ABB RAPID module: RsTempModule.mod

MODULE RsTempModule
    LOCAL CONST robtarget Target_10:=[[1336,100,940],[0.180407894,-0.26458531,0.050458418,0.945992364],[0,0,0,0],[9E+09,9E+09,9E+09,9E+09,9E+09,9E+09]];
    LOCAL CONST robtarget Target_20:=[[1131.146597498,-0.535735061,989.137836506],[0.652828066,-0.271690111,-0.271690111,-0.652828066],[0,0,0,0],[9E+09,9E+09,9E+09,9E+09,9E+09,9E+09]];
    LOCAL CONST robtarget Target_30:=[[1336,-49,1090],[0.946229257,-0.045801741,0.154506016,0.280500063],[0,0,0,0],[9E+09,9E+09,9E+09,9E+09,9E+09,9E+09]];
PROC RsTempPath()
        MoveC Target_20,Target_30,v1000,z100,tool0\WObj:=wobj0;
ENDPROC

ENDMODULE
